Staubli VAL3: moveSpinner.pgx

program moveSpinner()
begin
  movej(spinnerPosition,flange,mFastMov)
  waitEndMove()
  message="moveSpinner:done"
  taskCreate "sendStatus",100,sendStatus()
  taskKill("moveSpinner")
end
